FUNCTION_BLOCK PUBLIC FB_AirConditioning
VAR_OUTPUT
	bActive			: BOOL;
	lrTemperature	: LREAL;
END_VAR

METHOD PUBLIC Activate
bActive := TRUE;
END_METHOD

PROPERTY PUBLIC Activated : BOOL
GET
Activated := bActive;
END_GET
END_PROPERTY

METHOD PUBLIC Deactivate
bActive := false;
END_METHOD

METHOD PUBLIC SetTemperature : BOOL
VAR_INPUT
	lrNewTemperature	: LREAL;
END_VAR
lrTemperature := lrNewTemperature;
END_METHOD

PROPERTY PUBLIC Temperature : LREAL
GET
Temperature := lrTemperature;
END_GET
END_PROPERTY

END_FUNCTION_BLOCK

(* stored: Version 1.1.0.1, ProductVersion 3.1.4020.3
   POU FB_AirConditioning: Id {9d3aa5fb-75f3-46fa-8e76-d674e59fa53c}, SpecialFunc None
   Method Activate: Id {1a2fec03-c5e2-49d2-a4a1-00216e328eda}
   Property Activated: Id {0e2a419a-f906-4720-bd72-d3033aca54fb}
   Get Get: Id {7a7b69cf-468b-44cd-8277-7a1f46de03f6}
   Method Deactivate: Id {9c23aefa-366b-4734-af31-3dbe5cc4e27e}
   Method SetTemperature: Id {89d40da5-935c-42f7-aa47-6dc360b9ad3a}
   Property Temperature: Id {047500d1-4fdb-469e-adee-34ed6faba710}
   Get Get: Id {f17493df-ca76-438e-b178-a1124cd31740} *)
